FUNCTION_BLOCK ProductOrders
  (* Standard: 61499-2 *)
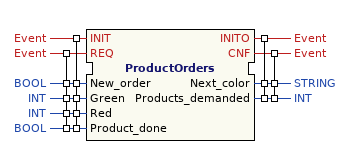
  EVENT_INPUT
    INIT WITH New_order, Green, Red, Product_done;
    REQ WITH Green, New_order, Product_done, Red;
  END_EVENT
  EVENT_OUTPUT
    INITO WITH Next_color, Products_demanded;
    CNF WITH Next_color, Products_demanded;
  END_EVENT
  VAR_INPUT
    New_order : BOOL;
    Green : INT;
    Red : INT;
    Product_done : BOOL;
  END_VAR
  VAR_OUTPUT
    Next_color : STRING;
    Products_demanded : INT;
  END_VAR
  VAR
    Green_count : INT;
    Red_count : INT;
    Product_count : INT;
  END_VAR
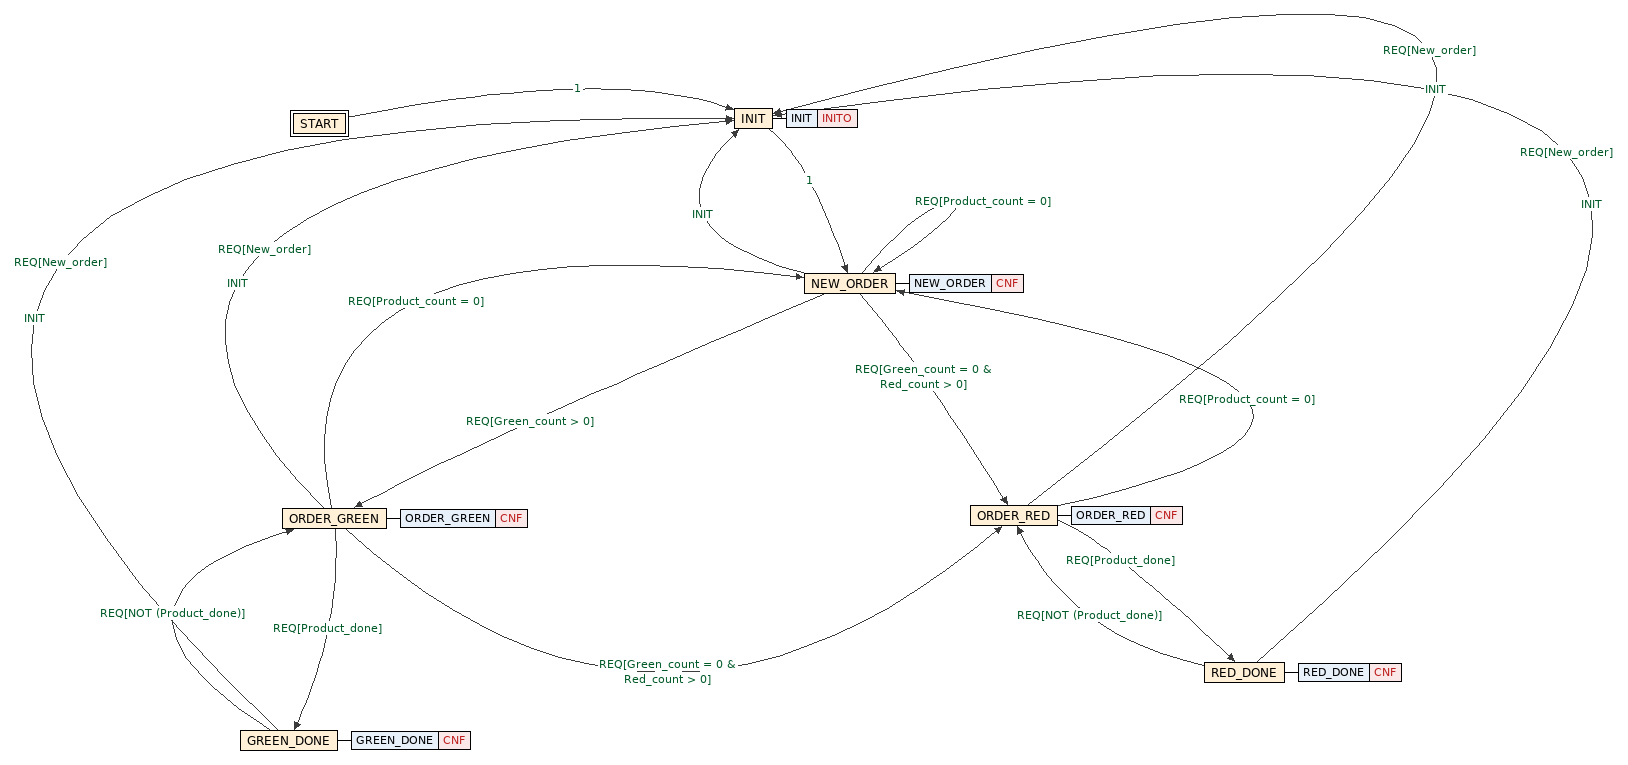
  EC_STATES
    START;
    INIT : INIT -> INITO;
    NEW_ORDER : NEW_ORDER -> CNF;
    ORDER_GREEN : ORDER_GREEN -> CNF;
    ORDER_RED : ORDER_RED -> CNF;
    GREEN_DONE : GREEN_DONE -> CNF;
    RED_DONE : RED_DONE -> CNF;
  END_STATES
  EC_TRANSITIONS
    START TO INIT := 1;
    INIT TO NEW_ORDER := 1;
    NEW_ORDER TO ORDER_GREEN := REQ[Green_count > 0];
    NEW_ORDER TO ORDER_RED := REQ[Green_count = 0 & Red_count > 0];
    NEW_ORDER TO NEW_ORDER := REQ[Product_count = 0];
    ORDER_GREEN TO ORDER_RED := REQ[Green_count = 0 & Red_count > 0];
    ORDER_GREEN TO NEW_ORDER := REQ[Product_count = 0];
    ORDER_RED TO NEW_ORDER := REQ[Product_count = 0];
    ORDER_GREEN TO INIT := INIT;
    ORDER_GREEN TO INIT := REQ[New_order];
    ORDER_RED TO INIT := INIT;
    ORDER_RED TO INIT := REQ[New_order];
    NEW_ORDER TO INIT := INIT;
    ORDER_GREEN TO GREEN_DONE := REQ[Product_done];
    GREEN_DONE TO ORDER_GREEN := REQ[NOT (Product_done)];
    ORDER_RED TO RED_DONE := REQ[Product_done];
    RED_DONE TO ORDER_RED := REQ[NOT (Product_done)];
    GREEN_DONE TO INIT := INIT;
    GREEN_DONE TO INIT := REQ[New_order];
    RED_DONE TO INIT := INIT;
    RED_DONE TO INIT := REQ[New_order];
  END_TRANSITIONS
  ALGORITHM INIT IN ST:
Green_count := 0;&#10;Red_count := 0;&#10;Product_count := 0;&#10;Products_demanded := 0;&#10;Next_color := 'NONE';&#10;
  END_ALGORITHM
  ALGORITHM NEW_ORDER IN ST:
Red_count := Red;&#10;Green_count := Green;&#10;Product_count := Red_count + Green_count;&#10;Products_demanded := Product_count;&#10;Next_color := 'NONE';&#10;
  END_ALGORITHM
  ALGORITHM ORDER_GREEN IN ST:
Products_demanded := Product_count;&#10;Next_color := 'GREEN';&#10;
  END_ALGORITHM
  ALGORITHM ORDER_RED IN ST:
Products_demanded := Product_count;&#10;Next_color := 'RED';&#10;
  END_ALGORITHM
  ALGORITHM GREEN_DONE IN ST:
Green_count := Green_count - 1;&#10;Product_count := Green_count + Red_count;&#10;Products_demanded := Product_count;&#10;Next_color := 'GREEN';&#10;
  END_ALGORITHM
  ALGORITHM RED_DONE IN ST:
Red_count := Red_count - 1;&#10;Product_count := Green_count + Red_count;&#10;Products_demanded := Product_count;&#10;Next_color := 'RED';&#10;
  END_ALGORITHM
END_FUNCTION_BLOCK
